{attribute 'GeneratedUsingTerminal: EL3314-0030-0021'}
{attribute addProperty BoxType "EL3314-0030-0021"}
{attribute addProperty Id "UnderrangeBOOL1OverrangeBOOL1ErrorBOOL1TxPDO_StateBOOL1TxPDO_ToggleBOOL1"}
{attribute addProperty CRC "1757626009"}
{attribute addProperty Size "5"}
TYPE Status_68C33E99 :
STRUCT
	{attribute addProperty Name "Underrange"}
	Underrange : BOOL;
	{attribute addProperty Name "Overrange"}
	Overrange : BOOL;
	{attribute addProperty Name "Error"}
	Error : BOOL;
	{attribute addProperty Name "TxPDO_State"}
	TxPDO_State : BOOL;
	{attribute addProperty Name "TxPDO_Toggle"}
	TxPDO_Toggle : BOOL;
END_STRUCT
END_TYPE

(* stored: Version 1.2.0.0, ProductVersion 3.1.4024.9
   DUT Status_68C33E99: Id {112a0de8-6da2-412c-95ec-1b7f0c41e6e9} *)
